// This function has been automatically generated from the project information.
{attribute 'signature_flag' := '1073741824'}
{attribute 'TcGenerated'}
{attribute 'no-analysis'}
FUNCTION F_GetTitle : WSTRING
VAR_INPUT
	
END_VAR

F_GetTitle := "CNM_AbstractObject";

END_FUNCTION

(* stored: Version 1.1.0.1, ProductVersion 3.1.4026.7
   POU F_GetTitle: Id {5b39faaf-3fe5-4a46-92cc-430951517afe}, SpecialFunc None *)
